INTERFACE I_AnimalTraits EXTENDS I_AnimalFamily

METHOD DietType : BOOL
VAR_INPUT
END_VAR
END_METHOD

METHOD IsDangerous : BOOL
VAR_INPUT
END_VAR
END_METHOD

PROPERTY RevivalTime : TIME
GET
END_GET
SET
END_SET
END_PROPERTY

END_INTERFACE

(* stored: Version 1.1.0.1, ProductVersion 3.1.4024.16
   Itf I_AnimalTraits: Id {156cb202-02be-41b8-93af-e2b80bb59c83}
   Method DietType: Id {b3977abb-e730-40c0-89df-bc0ea2b290a4}
   Method IsDangerous: Id {44900d0e-acb6-4573-8f96-0e64f8abf7c2}
   Property RevivalTime: Id {90c5d45b-1850-47a6-83a5-53d48f3debdb}
   Get Get: Id {3e8843ea-d75e-4ea6-8f09-b16d65419ac4}
   Set Set: Id {aa7d94ba-6eb3-45cb-a222-797cf73a86e0} *)
